# EPICS substitutions: ek9000App/Db/EL3201.substitutions
file EL3201.template
{ 	pattern
	{
		TERMINAL,

	}
	{
	}
}

	}
	{
	}
}
